{attribute addProperty BoxType "EL6201-0000-0017"}
{attribute addProperty Id "Slave_4A_DO0BIT10.12525Slave_4A_DO1BIT10.12526Slave_4A_DO2BIT10.12527Slave_4A_DO3BIT10.12528Slave_4B_DO0BIT10.12529Slave_4B_DO1BIT10.12530Slave_4B_DO2BIT10.12531Slave_4B_DO3BIT10.12532"}
{attribute addProperty CRC "2730831755"}
{attribute addProperty SizeInBites "8"}
{attribute addProperty SizeInBytes "1"}
TYPE Slave_4_Outputs_A2C52F8B :
STRUCT
	{attribute addProperty Name "Slave_4A_DO0"}
	Slave_4A_DO0 : BIT;
	{attribute addProperty Name "Slave_4A_DO1"}
	Slave_4A_DO1 : BIT;
	{attribute addProperty Name "Slave_4A_DO2"}
	Slave_4A_DO2 : BIT;
	{attribute addProperty Name "Slave_4A_DO3"}
	Slave_4A_DO3 : BIT;
	{attribute addProperty Name "Slave_4B_DO0"}
	Slave_4B_DO0 : BIT;
	{attribute addProperty Name "Slave_4B_DO1"}
	Slave_4B_DO1 : BIT;
	{attribute addProperty Name "Slave_4B_DO2"}
	Slave_4B_DO2 : BIT;
	{attribute addProperty Name "Slave_4B_DO3"}
	Slave_4B_DO3 : BIT;
END_STRUCT
END_TYPE

(* stored: Version 1.2.0.0, ProductVersion 3.1.4024.9
   DUT Slave_4_Outputs_A2C52F8B: Id {ede7a48c-12d0-429c-bd1a-103d8578745a} *)
